Fanuc KAREL source: kb00150.KL

-- PROVISIONAL review KL for V940-1; original PC SHA256 334233150b0f05ce357463cc1a8ad16beafa920f86aa74e1f23ff47982f64b72
-- Incomplete behavior may be omitted. Consult companion uncertainty JSON. Do not deploy.
PROGRAM KB00150
%NOLOCKGROUP
BEGIN
  -- V9_ZERO_TABLE_METADATA_HINT layout=0002_ascii; no indexed target words; source/name/runtime held
  -- UNRESOLVED_PC offsets 5-14; opcodes 3F,75
  -- UNRESOLVED_PC offsets 19-28; opcodes 3F,75
  -- UNRESOLVED_PC offsets 33-42; opcodes 3F,75
  -- UNRESOLVED_PC offsets 47-56; opcodes 3F,75
  -- UNRESOLVED_PC offsets 61-68; opcodes 9D,23
  -- UNRESOLVED_PC offsets 73-115; opcodes 27,22,2A,22,2A,22,2A,22,2A,22,31
  -- UNRESOLVED_PC offsets 120-124; opcodes 7F
END KB00150
